FUNCTION_BLOCK FB_FTP_FindAllPartProgram 
VAR_INPUT
	Execute 	: BOOL;
	sNetId		: STRING;
	sPathName	: STRING;
	Username	: STRING;
	Password	: STRING;
	sHost		: STRING;
END_VAR
VAR_OUTPUT
	Busy 		: BOOL;
	Done 		: BOOL;
	Error 		: BOOL;
	ErrorID 	: DINT;
	ErrorSubID 	: UDINT;
    FileList    : ARRAY [0..99] OF STRING;
    Items       : UDINT;
END_VAR
VAR
	iState 			: DINT := -1;
	i 				: USINT;
	RTRIG_Execute 	: R_TRIG;
	fbFTP_Open		: FB_FTP_Open;
	fbFTP_Close		: FB_FTP_Close;
	fbFTP_Search	: FB_FTP_FileList;
	TON_Timeout		: TON;
    TempFileList    : ARRAY [0..99] OF STRING;
    TempItems       : UDINT;
END_VAR

TON_Timeout(IN := Busy, PT := T#20S);
IF TON_Timeout.Q THEN
	
	iState := 1999;
END_IF

RTRIG_Execute(CLK := Execute);
IF(RTRIG_Execute.Q) THEN
	Done := FALSE;
	i := 0;
	ErrorID := 0;
	ErrorSubID := 0;	
	
	iState := 0;
ELSIF NOT Execute AND NOT Busy THEN
	Busy			:= FALSE;
	Done			:= FALSE;
	Error			:= FALSE;
	
	iState := -1;
END_IF

CASE iState OF
	-1:
		;
		
	0:
		Busy := TRUE;
		fbFTP_Open.bExecute := TRUE;
		iState := 10;
		
	10:
		fbFTP_Open.bExecute := FALSE; 
        IF NOT fbFTP_Open.bBusy THEN 
        	IF fbFTP_Open.bError THEN 
            	ErrorSubID := fbFTP_Open.nErrId; 
                iState := 1010;
               ELSE 
                 	iState := 20;
               END_IF 
          END_IF
		
	20:
		fbFTP_Search.bExecute := TRUE;
		iState := 30;
			
	30:
        fbFTP_Search.bExecute := FALSE; 
        IF NOT fbFTP_Search.bBusy THEN 
        	IF fbFTP_Search.bError THEN 
            	ErrorSubID := fbFTP_Search.nErrId; 
                iState := 1030;
               ELSE 
				   Items := TempItems;
				   FileList := TempFileList;
				   
                 	iState := 990;
               END_IF 
          END_IF
		
	990:
		fbFTP_Close.bExecute := TRUE;
		iState := 991;
		
	991:
		fbFTP_Close.bExecute := FALSE; 
        IF NOT fbFTP_Close.bBusy THEN 
        	IF fbFTP_Close.bError THEN 
            	ErrorSubID := fbFTP_Close.nErrId; 
                iState := 1991;
               ELSE 
                 	iState := 999;
               END_IF 
          END_IF	

	999:
		Busy	 			:= FALSE;
		Done				:= TRUE;
	
		iState := -1;	
END_CASE

IF(iState > 999) THEN
	Error 	:= TRUE;
	ErrorID := iState;
	Busy 	:= FALSE;
ELSE
	Error := FALSE;
END_IF

A_Call();

ACTION A_Call:
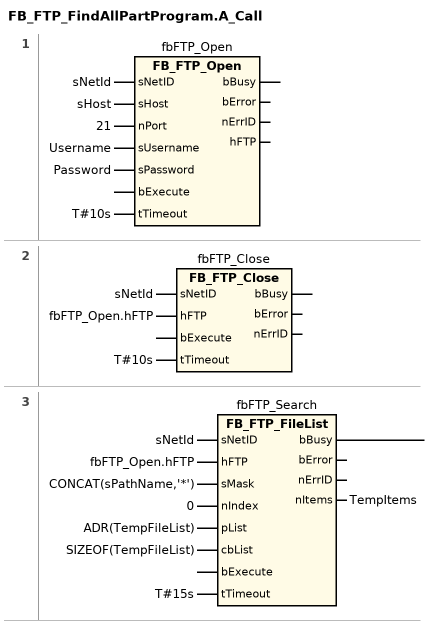
// NETWORK 1
fbFTP_Open(
    sNetID := sNetId,
    sHost := sHost,
    nPort := 21,
    sUsername := Username,
    sPassword := Password,
    tTimeout := T#10s); // FB_FTP_Open

// NETWORK 2
fbFTP_Close(sNetID := sNetId, hFTP := fbFTP_Open.hFTP, tTimeout := T#10s); // FB_FTP_Close

// NETWORK 3
fbFTP_Search(
    sNetID := sNetId,
    hFTP := fbFTP_Open.hFTP,
    sMask := CONCAT(sPathName,'*'),
    nIndex := 0,
    pList := ADR(TempFileList),
    cbList := SIZEOF(TempFileList),
    tTimeout := T#15s,
    nItems => TempItems); // FB_FTP_FileList
END_ACTION

END_FUNCTION_BLOCK

(* stored: Version 1.1.0.1, ProductVersion 3.1.4024.13
   POU FB_FTP_FindAllPartProgram: Id {dee1be80-9aa7-4f09-8c7e-6d4d0d4d3d97}, SpecialFunc None
   Action A_Call: Id {42c4b01c-6542-4a84-a3b3-3cfe72ceecf2} *)
